FUNCTION PID 
VAR_INPUT
	enable: BOOL;
	
END_VAR
VAR_IN_OUT
	e0, e1, e2: REAL;
	u0, u1: REAL;
	p, i, d: REAL;
	set, mea: REAL;
	stime: REAL;
	
END_VAR
VAR
END_VAR

IF (enable = TRUE) THEN
	e2 := e1;
	e1 := e0;
	e0 := set - mea;
	u1 := u0;
	u0 := u1 + p*(e0 - e1) + i*stime*(e0 + e1)/2.0 + d*(e0 - 2*e1 + e2)/stime;
END_IF

END_FUNCTION

(* stored: Version 1.1.0.1, ProductVersion 3.1.4024.3
   POU PID: Id {3be49269-d286-45a5-b12d-a57be8ebfef9}, SpecialFunc None *)
